{attribute addProperty BoxType "EK1100-0000-0018"}
{attribute addProperty Id "Beckhoff_EQ1xxxEK1122Beckhoff_EQ1xxxEK1122_FDDE2AD855469.25"}
{attribute addProperty CRC "2184047323"}
{attribute addProperty SizeInBites "554"}
{attribute addProperty SizeInBytes "69.25"}
TYPE Beckhoff_EQ1xxx_822DEADB EXTENDS EK1100_179A0949 :
STRUCT
	{attribute addProperty Name "Beckhoff_EQ1xxxEK1122"}
	Beckhoff_EQ1xxxEK1122 : Beckhoff_EQ1xxxEK1122_FDDE2AD8;
END_STRUCT
END_TYPE

(* stored: Version 1.2.0.0, ProductVersion 3.1.4024.9
   DUT Beckhoff_EQ1xxx_822DEADB: Id {c739aa75-8f62-414d-b8de-03d6de6a387c} *)
